FUNCTION_BLOCK TYPE_SERIALIZER (* Basic FB with empty ECC *)
  (* Standard: 61499-2 *)
  (* Version 1.0, 2023-04-21, valentinnodan *)
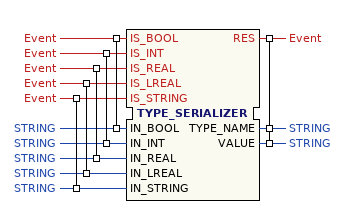
  EVENT_INPUT
    IS_BOOL WITH IN_BOOL;
    IS_INT WITH IN_INT;
    IS_REAL WITH IN_REAL;
    IS_LREAL WITH IN_LREAL;
    IS_STRING WITH IN_STRING;
  END_EVENT
  EVENT_OUTPUT
    RES WITH TYPE_NAME, VALUE;
  END_EVENT
  VAR_INPUT
    IN_BOOL : STRING;
    IN_INT : STRING;
    IN_REAL : STRING;
    IN_LREAL : STRING;
    IN_STRING : STRING;
  END_VAR
  VAR_OUTPUT
    TYPE_NAME : STRING;
    VALUE : STRING;
  END_VAR
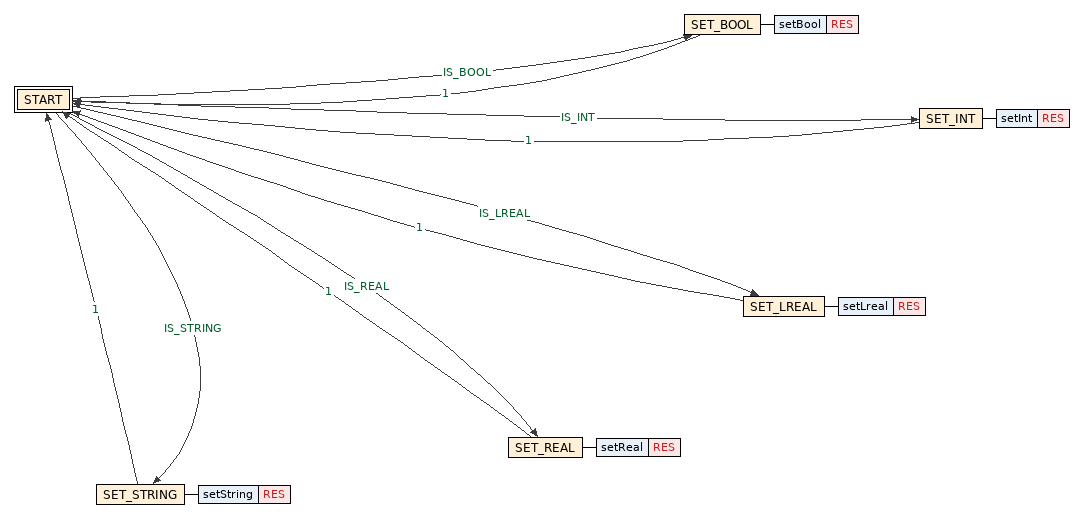
  EC_STATES
    START; (* Initial State *)
    SET_BOOL : setBool -> RES;
    SET_INT : setInt -> RES;
    SET_LREAL : setLreal -> RES;
    SET_REAL : setReal -> RES;
    SET_STRING : setString -> RES;
  END_STATES
  EC_TRANSITIONS
    START TO SET_STRING := IS_STRING;
    SET_STRING TO START := 1;
    START TO SET_REAL := IS_REAL;
    SET_REAL TO START := 1;
    START TO SET_LREAL := IS_LREAL;
    SET_LREAL TO START := 1;
    START TO SET_BOOL := IS_BOOL;
    SET_BOOL TO START := 1;
    START TO SET_INT := IS_INT;
    SET_INT TO START := 1;
  END_TRANSITIONS
  ALGORITHM setBool IN ST:
TYPE_NAME := 'BOOL';
VALUE := IN_BOOL;
  END_ALGORITHM
  ALGORITHM setInt IN ST:
TYPE_NAME := 'INT';
VALUE := IN_INT;
  END_ALGORITHM
  ALGORITHM setReal IN ST:
TYPE_NAME := 'REAL';
VALUE := IN_REAL;
  END_ALGORITHM
  ALGORITHM setLreal IN ST:
TYPE_NAME := 'LREAL';
VALUE := IN_LREAL;
  END_ALGORITHM
  ALGORITHM setString IN ST:
TYPE_NAME := 'STRING';
VALUE := IN_STRING;
  END_ALGORITHM
END_FUNCTION_BLOCK
